// TIA Portal project "Elektriksel Kilitleme" (V18)

(* hardware
DEVICE "S7-1200 station_1"  S7-1200 Station
   slot 0: "Rack_0"  S7-1200 Rack  Rack  V1.0
   slot 1: "PLC_1"  CPU 1212C DC/DC/DC  6ES7 212-1AE40-0XB0  V4.6
*)

// ===== PLC "PLC_1"  CPU 1212C DC/DC/DC =====

VAR_GLOBAL   // PLC tag table "Default tag table"
   "ILERI START BUT" AT %I0.0 : Bool;
   "GERI START BUT" AT %I0.1 : Bool;
   "STOP BUT" AT %I0.2 : Bool;
   "ILERI KONT" AT %Q0.0 : Bool;
   "GERI KONT" AT %Q0.1 : Bool;
   "ILERI LAMBA" AT %Q0.2 : Bool;
   "GERI LAMBA" AT %Q0.3 : Bool;
   "STOP LAMBA" AT %Q0.4 : Bool;
END_VAR

ORGANIZATION_BLOCK "Main"   // OB1, LAD, ProgramCycle
TITLE = "Main Program Sweep (Cycle)"
{ S7_Optimized_Access := 'TRUE' }
VERSION : 0.1
   VAR_INPUT
      Initial_Call : Bool;   // Initial call of this OB
      Remanence : Bool;   // =True, if remanent data are available
   END_VAR
   VAR_TEMP   // added for the SCL form of the ladder/FBD networks
      _w1 : Bool;
   END_VAR
BEGIN

REGION Network 1: İLERİ YÖN KONTROLÜ VE ELEKTRİKSEL KİLİTLEME
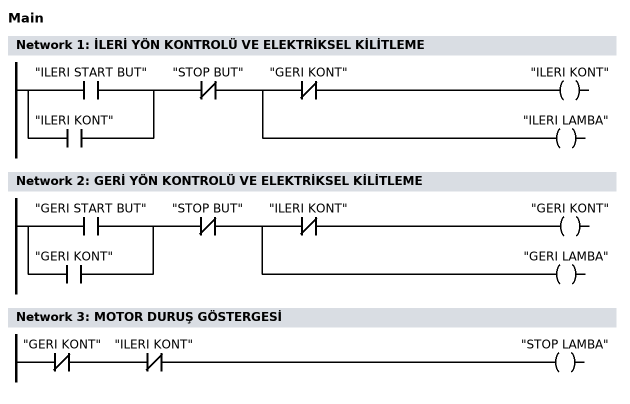
   RUNG wire#powerrail
      Contact( "ILERI START BUT" )
      wire#w1
      I_Contact( "STOP BUT" )
      wire#w2
      I_Contact( "GERI KONT" )
      Coil( "ILERI KONT" )
   END_RUNG
   RUNG wire#powerrail
      Contact( "ILERI KONT" )
   END_RUNG wire#w1
   RUNG wire#w2
      Coil( "ILERI LAMBA" )
   END_RUNG
   // the same network as SCL:
   #_w1 := ("ILERI START BUT" OR "ILERI KONT") AND NOT "STOP BUT";
   "ILERI KONT" := #_w1 AND NOT "GERI KONT";
   "ILERI LAMBA" := #_w1;
END_REGION

REGION Network 2: GERİ YÖN KONTROLÜ VE ELEKTRİKSEL KİLİTLEME
   RUNG wire#powerrail
      Contact( "GERI START BUT" )
      wire#w1
      I_Contact( "STOP BUT" )
      wire#w2
      I_Contact( "ILERI KONT" )
      Coil( "GERI KONT" )
   END_RUNG
   RUNG wire#powerrail
      Contact( "GERI KONT" )
   END_RUNG wire#w1
   RUNG wire#w2
      Coil( "GERI LAMBA" )
   END_RUNG
   // the same network as SCL:
   #_w1 := ("GERI START BUT" OR "GERI KONT") AND NOT "STOP BUT";
   "GERI KONT" := #_w1 AND NOT "ILERI KONT";
   "GERI LAMBA" := #_w1;
END_REGION

REGION Network 3: MOTOR DURUŞ GÖSTERGESİ
   RUNG wire#powerrail
      I_Contact( "GERI KONT" )
      I_Contact( "ILERI KONT" )
      Coil( "STOP LAMBA" )
   END_RUNG
   // the same network as SCL:
   "STOP LAMBA" := NOT "GERI KONT" AND NOT "ILERI KONT";
END_REGION
END_ORGANIZATION_BLOCK